// TIA Portal project "FactoryIO_Template_S7-1200_V15_V19_1" (V19)
// Vorlageprojekt für das Buch mit Zielsystem S7-1200

(* hardware
DEVICE "S7-1200-Station_1"  S7-1200 Station
   slot 0: "Baugruppenträger_0"  Rack  V1.0
   slot 1: "PLC_1"  CPU 1211C DC/DC/DC  6ES7 211-1AE40-0XB0  V4.1
*)

// ===== PLC "PLC_1"  CPU 1211C DC/DC/DC =====

VAR_GLOBAL   // PLC tag table "Standard-Variablentabelle"
   "KONVEYÖR 1" AT %A0.0 : Bool;
   "START" AT %E0.0 : Bool;
   "STOP" AT %E0.1 : Bool;
   "Tag_4" AT %M0.0 : Bool;
   "KONVEYÖR 2" AT %Q0.1 : Bool;
   "Tag_6" AT %M0.1 : Bool;
   "RESET" AT %I0.2 : Bool;
   "ÇIKIŞ SENSÖRÜ" AT %I0.3 : Bool;
   "KONVEYÖR 3" AT %Q0.2 : Bool;
   "KONVEYÖR 4" AT %Q0.3 : Bool;
   "Tag_11" AT %M0.2 : Bool;
   "SİSTEM START MEMORY" AT %M10.0 : Bool;
   "VISION SENSOR" AT %ID30 : DInt;
   "TETİK_1" AT %M30.2 : Bool;
   "KONVEYÖR 1 STOP" AT %M14.0 : Bool;
   "TETİK_2" AT %M30.3 : Bool;
   "ÇIKIŞ KONVEYÖRÜ" AT %Q0.7 : Bool;
   "KONVEYÖR 2 DÖN" AT %Q0.4 : Bool;
   "TETİK_3" AT %M20.6 : Bool;
   "TETİK_4" AT %M19.0 : Bool;
   "KONVEYÖR 3 DÖN" AT %Q0.5 : Bool;
   "KONVEYÖR 4 DÖN" AT %Q0.6 : Bool;
   "TETİK_5" AT %M12.5 : Bool;
   "KUTU SAYISI" AT %MW28 : Int;
   "SAYAÇ" AT %QD30 : DWord;
END_VAR

FUNCTION "MHJ-PLC-Lab-Function-S71200" : Void   // FC9000, SCL
{ S7_Optimized_Access := 'TRUE' }
VERSION : 0.1
   VAR_TEMP
      rdTimeReturn : Int;
      outputTime : DTL;
      SyncVal : Byte;
      forVal : Int;
      forVal_2 : Int;
      Value : Byte;
   END_VAR
   VAR CONSTANT
      CompVal : Byte := 16#34;
      Value_01 : Byte := 16#11;
      Value_01_DW : DWord := 16#A165_D992;
      Value_02_DW : DWord := 16#58BE_4401;
   END_VAR
BEGIN

   #Value:=PEEK(area := 16#82,
        dbNumber := 0,
        byteOffset := 511);
   #Value := #Value + 1;

   POKE(area := 16#82,
        dbNumber := 0,
        byteOffset := 511,
        value := #Value);

   POKE(area:=16#81,
        dbNumber:=0,
        byteOffset:=1016,
        value:=#Value_01_DW);
   POKE(area := 16#81,
        dbNumber := 0,
        byteOffset := 1020,
        value := #Value_02_DW);

   POKE(area := 16#81,
        dbNumber := 0,
        byteOffset := 511,
        value := B#16#00);

   FOR #forVal := 0 TO 120 DO
       FOR #forVal_2:=0 TO 10 DO
           #rdTimeReturn:=RD_SYS_T(#outputTime);
           #rdTimeReturn := WR_SYS_T(#outputTime);
           #rdTimeReturn := RD_SYS_T(#outputTime);
           #rdTimeReturn := WR_SYS_T(#outputTime);
       END_FOR;
       #SyncVal:= PEEK(area := 16#81,
                      dbNumber := 0,
                      byteOffset := 511);
       IF #SyncVal = #CompVal THEN
          GOTO M_1;
       END_IF;
   END_FOR;
   RETURN;

   M_1:
   POKE(area := 16#81,
        dbNumber := 0,
        byteOffset := 511,
        value := B#16#0);
END_FUNCTION

ORGANIZATION_BLOCK "Main"   // OB1, LAD, ProgramCycle
TITLE = "Main Program Sweep (Cycle)"
{ S7_Optimized_Access := 'TRUE' }
VERSION : 0.1
   VAR_INPUT
      Initial_Call : Bool;   // Initial call of this OB
      Remanence : Bool;   // =True, if remanent data are available
   END_VAR
   VAR_TEMP   // added for the SCL form of the ladder/FBD networks
      _w1 : Bool;
      _w2 : Bool;
      _w3 : Bool;
      _w4 : Bool;
   END_VAR
BEGIN

REGION Network 1: Konnektierungsbaustein für PLC-Lab
   // Im Netzwerk 1 wird der Konnektierungsbaustein für PLC-Lab aufgerufen.
   // Dieser Aufruf darf nicht entfernt werden!
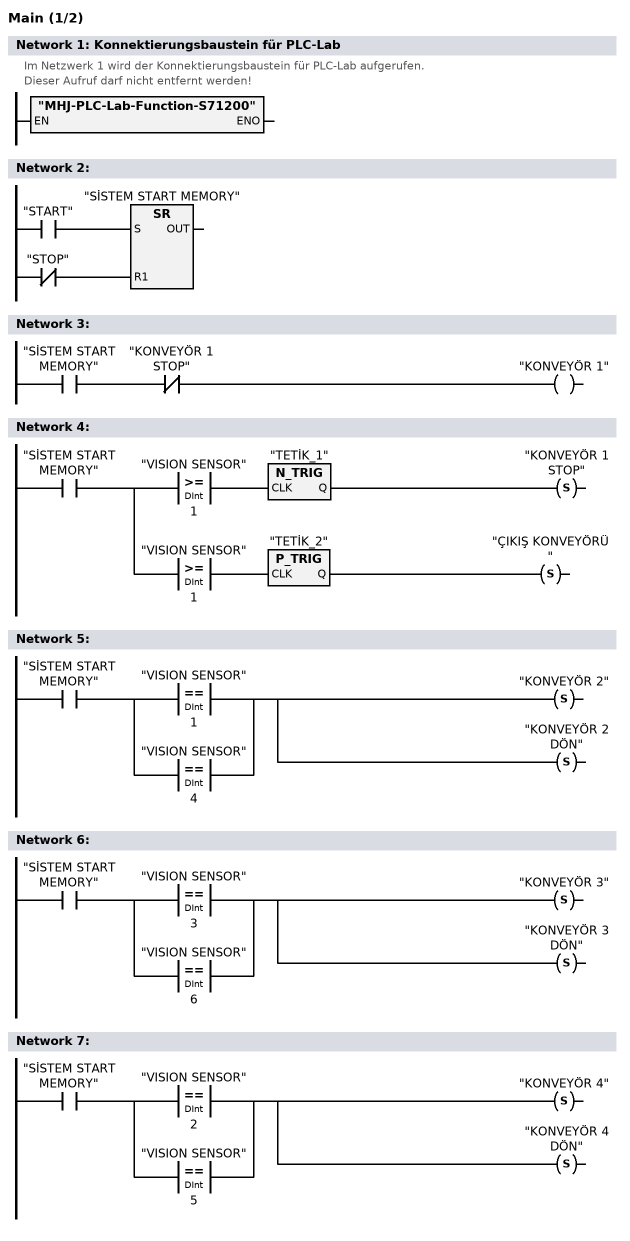
   RUNG wire#powerrail
      "MHJ-PLC-Lab-Function-S71200"()
   END_RUNG
   // the same network as SCL:
   "MHJ-PLC-Lab-Function-S71200"();
END_REGION

REGION Network 2
   RUNG wire#powerrail
      Contact( "START" )
      S_SR(operand := "SİSTEM START MEMORY", r1 := wire#w1)
   END_RUNG
   RUNG wire#powerrail
      I_Contact( "STOP" )
   END_RUNG wire#w1
   // the same network as SCL:
   IF "START" THEN
       "SİSTEM START MEMORY" := TRUE;   // SR flip-flop
   END_IF;
   IF NOT "STOP" THEN "SİSTEM START MEMORY" := FALSE; END_IF;
END_REGION

REGION Network 3
   RUNG wire#powerrail
      Contact( "SİSTEM START MEMORY" )
      I_Contact( "KONVEYÖR 1 STOP" )
      Coil( "KONVEYÖR 1" )
   END_RUNG
   // the same network as SCL:
   "KONVEYÖR 1" := "SİSTEM START MEMORY" AND NOT "KONVEYÖR 1 STOP";
END_REGION

REGION Network 4
   RUNG wire#powerrail
      Contact( "SİSTEM START MEMORY" )
      wire#w1
      { S7_Templates := "SrcType := DInt" } GE_Contact(in1 := "VISION SENSOR", in2 := 1)
      N_Trig( "TETİK_1" )
      S_Coil( "KONVEYÖR 1 STOP" )
   END_RUNG
   RUNG wire#w1
      { S7_Templates := "SrcType := DInt" } GE_Contact(in1 := "VISION SENSOR", in2 := 1)
      P_Trig( "TETİK_2" )
      S_Coil( "ÇIKIŞ KONVEYÖRÜ" )
   END_RUNG
   // the same network as SCL:
   #_w1 := "SİSTEM START MEMORY" AND ("VISION SENSOR" >= 1);
   #_w2 := NOT #_w1 AND "TETİK_1";   // falling edge
   "TETİK_1" := #_w1;
   IF #_w2 THEN "KONVEYÖR 1 STOP" := TRUE; END_IF;
   #_w3 := "SİSTEM START MEMORY" AND ("VISION SENSOR" >= 1);
   #_w4 := #_w3 AND NOT "TETİK_2";   // rising edge
   "TETİK_2" := #_w3;
   IF #_w4 THEN "ÇIKIŞ KONVEYÖRÜ" := TRUE; END_IF;
END_REGION

REGION Network 5
   RUNG wire#powerrail
      Contact( "SİSTEM START MEMORY" )
      wire#w1
      { S7_Templates := "SrcType := DInt" } EQ_Contact(in1 := "VISION SENSOR", in2 := 1)
      wire#w2
      S_Coil( "KONVEYÖR 2" )
   END_RUNG
   RUNG wire#w1
      { S7_Templates := "SrcType := DInt" } EQ_Contact(in1 := "VISION SENSOR", in2 := 4)
   END_RUNG wire#w2
   RUNG wire#w2
      S_Coil( "KONVEYÖR 2 DÖN" )
   END_RUNG
   // the same network as SCL:
   IF "SİSTEM START MEMORY" AND (("VISION SENSOR" = 1) OR ("VISION SENSOR" = 4)) THEN
       "KONVEYÖR 2" := TRUE;
       "KONVEYÖR 2 DÖN" := TRUE;
   END_IF;
END_REGION

REGION Network 6
   RUNG wire#powerrail
      Contact( "SİSTEM START MEMORY" )
      wire#w1
      { S7_Templates := "SrcType := DInt" } EQ_Contact(in1 := "VISION SENSOR", in2 := 3)
      wire#w2
      S_Coil( "KONVEYÖR 3" )
   END_RUNG
   RUNG wire#w1
      { S7_Templates := "SrcType := DInt" } EQ_Contact(in1 := "VISION SENSOR", in2 := 6)
   END_RUNG wire#w2
   RUNG wire#w2
      S_Coil( "KONVEYÖR 3 DÖN" )
   END_RUNG
   // the same network as SCL:
   IF "SİSTEM START MEMORY" AND (("VISION SENSOR" = 3) OR ("VISION SENSOR" = 6)) THEN
       "KONVEYÖR 3" := TRUE;
       "KONVEYÖR 3 DÖN" := TRUE;
   END_IF;
END_REGION

REGION Network 7
   RUNG wire#powerrail
      Contact( "SİSTEM START MEMORY" )
      wire#w1
      { S7_Templates := "SrcType := DInt" } EQ_Contact(in1 := "VISION SENSOR", in2 := 2)
      wire#w2
      S_Coil( "KONVEYÖR 4" )
   END_RUNG
   RUNG wire#w1
      { S7_Templates := "SrcType := DInt" } EQ_Contact(in1 := "VISION SENSOR", in2 := 5)
   END_RUNG wire#w2
   RUNG wire#w2
      S_Coil( "KONVEYÖR 4 DÖN" )
   END_RUNG
   // the same network as SCL:
   IF "SİSTEM START MEMORY" AND (("VISION SENSOR" = 2) OR ("VISION SENSOR" = 5)) THEN
       "KONVEYÖR 4" := TRUE;
       "KONVEYÖR 4 DÖN" := TRUE;
   END_IF;
END_REGION

REGION Network 8
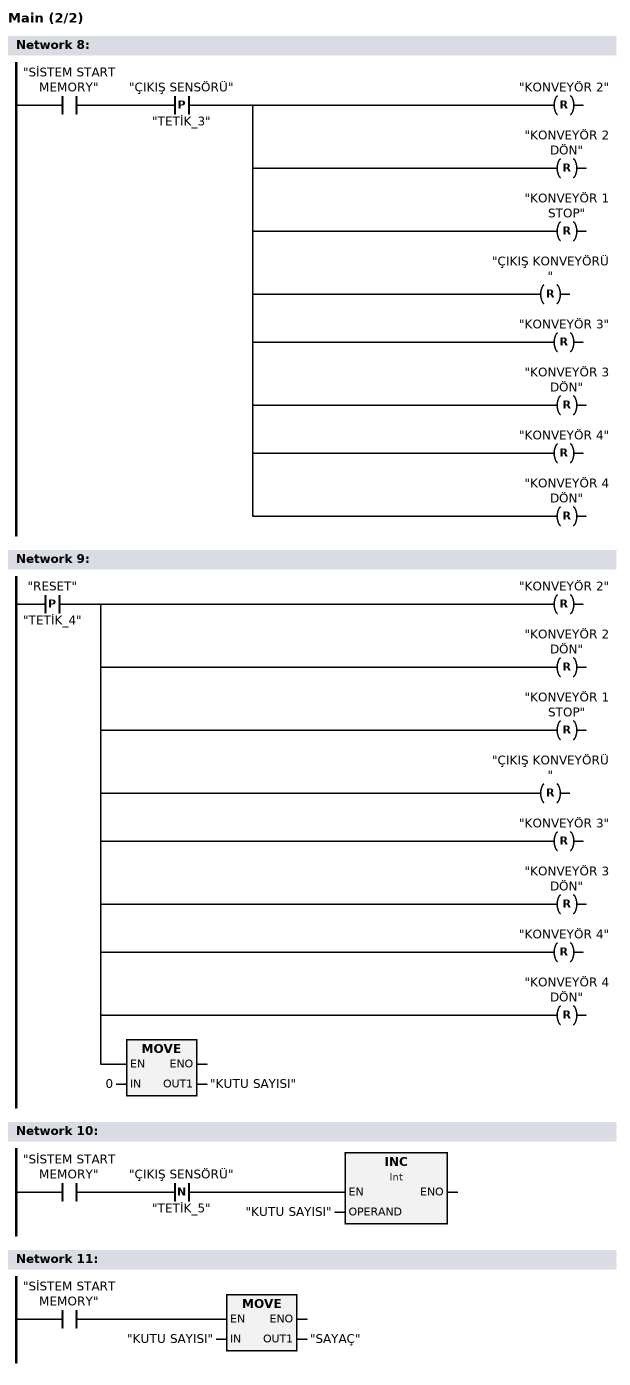
   RUNG wire#powerrail
      Contact( "SİSTEM START MEMORY" )
      P_Contact(operand := "ÇIKIŞ SENSÖRÜ", bit := "TETİK_3")
      wire#w1
      R_Coil( "KONVEYÖR 2" )
   END_RUNG
   RUNG wire#w1
      R_Coil( "KONVEYÖR 2 DÖN" )
   END_RUNG
   RUNG wire#w1
      R_Coil( "KONVEYÖR 1 STOP" )
   END_RUNG
   RUNG wire#w1
      R_Coil( "ÇIKIŞ KONVEYÖRÜ" )
   END_RUNG
   RUNG wire#w1
      R_Coil( "KONVEYÖR 3" )
   END_RUNG
   RUNG wire#w1
      R_Coil( "KONVEYÖR 3 DÖN" )
   END_RUNG
   RUNG wire#w1
      R_Coil( "KONVEYÖR 4" )
   END_RUNG
   RUNG wire#w1
      R_Coil( "KONVEYÖR 4 DÖN" )
   END_RUNG
   // the same network as SCL:
   #_w1 := "SİSTEM START MEMORY" AND "ÇIKIŞ SENSÖRÜ" AND NOT "TETİK_3";   // rising edge of "ÇIKIŞ SENSÖRÜ"
   "TETİK_3" := "ÇIKIŞ SENSÖRÜ";
   IF #_w1 THEN
       "KONVEYÖR 2" := FALSE;
       "KONVEYÖR 2 DÖN" := FALSE;
       "KONVEYÖR 1 STOP" := FALSE;
       "ÇIKIŞ KONVEYÖRÜ" := FALSE;
       "KONVEYÖR 3" := FALSE;
       "KONVEYÖR 3 DÖN" := FALSE;
       "KONVEYÖR 4" := FALSE;
       "KONVEYÖR 4 DÖN" := FALSE;
   END_IF;
END_REGION

REGION Network 9
   RUNG wire#powerrail
      P_Contact(operand := "RESET", bit := "TETİK_4")
      wire#w1
      R_Coil( "KONVEYÖR 2" )
   END_RUNG
   RUNG wire#w1
      R_Coil( "KONVEYÖR 2 DÖN" )
   END_RUNG
   RUNG wire#w1
      R_Coil( "KONVEYÖR 1 STOP" )
   END_RUNG
   RUNG wire#w1
      R_Coil( "ÇIKIŞ KONVEYÖRÜ" )
   END_RUNG
   RUNG wire#w1
      R_Coil( "KONVEYÖR 3" )
   END_RUNG
   RUNG wire#w1
      R_Coil( "KONVEYÖR 3 DÖN" )
   END_RUNG
   RUNG wire#w1
      R_Coil( "KONVEYÖR 4" )
   END_RUNG
   RUNG wire#w1
      R_Coil( "KONVEYÖR 4 DÖN" )
   END_RUNG
   RUNG wire#w1
      Move(in := 0, out1 => "KUTU SAYISI")
   END_RUNG
   // the same network as SCL:
   #_w1 := "RESET" AND NOT "TETİK_4";   // rising edge of "RESET"
   "TETİK_4" := "RESET";
   IF #_w1 THEN
       "KONVEYÖR 2" := FALSE;
       "KONVEYÖR 2 DÖN" := FALSE;
       "KONVEYÖR 1 STOP" := FALSE;
       "ÇIKIŞ KONVEYÖRÜ" := FALSE;
       "KONVEYÖR 3" := FALSE;
       "KONVEYÖR 3 DÖN" := FALSE;
       "KONVEYÖR 4" := FALSE;
       "KONVEYÖR 4 DÖN" := FALSE;
       "KUTU SAYISI" := 0;
   END_IF;
END_REGION

REGION Network 10
   RUNG wire#powerrail
      Contact( "SİSTEM START MEMORY" )
      N_Contact(operand := "ÇIKIŞ SENSÖRÜ", bit := "TETİK_5")
      { S7_Templates := "DestType := Int" } Inc( "KUTU SAYISI" )
   END_RUNG
   // the same network as SCL:
   #_w1 := "SİSTEM START MEMORY" AND NOT "ÇIKIŞ SENSÖRÜ" AND "TETİK_5";   // falling edge of "ÇIKIŞ SENSÖRÜ"
   "TETİK_5" := "ÇIKIŞ SENSÖRÜ";
   IF #_w1 THEN "KUTU SAYISI" := "KUTU SAYISI" + 1; END_IF;
END_REGION

REGION Network 11
   RUNG wire#powerrail
      Contact( "SİSTEM START MEMORY" )
      Move(in := "KUTU SAYISI", out1 => "SAYAÇ")
   END_RUNG
   // the same network as SCL:
   IF "SİSTEM START MEMORY" THEN "SAYAÇ" := "KUTU SAYISI"; END_IF;
END_REGION
END_ORGANIZATION_BLOCK